{attribute 'qualified_only'}
{attribute 'strict'}
TYPE SubLevelCondition :
(
	ERROR,
	RUN
);
END_TYPE

(* stored: Version 1.1.0.1, ProductVersion 3.1.4024.12
   DUT SubLevelCondition: Id {d7d53af6-4e0f-455e-ba88-c24b90d2da98} *)
